// TIA Portal V17 export
// export: Created 2023-12-22T15:28:33.5067968Z, ExportSetting WithDefaults, DisplayName Totally Integrated Automation Portal, DisplayVersion V17, DisplayName TIA Portal Openness, DisplayVersion V17, DisplayName TIA Portal Version Control Interface, DisplayVersion V17, DisplayName STEP 7 Professional, DisplayVersion V17, DisplayName STEP 7 Safety, DisplayVersion V17, DisplayName WinCC Advanced, DisplayVersion V17
DATA_BLOCK "Support_DB"   // DB1000
{ S7_Optimized_Access := 'TRUE' }
VERSION : 0.1
// stored: AutoNumber false, DBAccessibleFromOPCUA true, IsOnlyStoredInLoadMemory false, IsRetainMemResEnabled false, IsWriteProtectedInAS false, MemoryReserve 100
   VAR
      DTR_Clean : Bool;   // Очистка DTR
      DTR_1 : Int;   // Data Transfer 1
      DTR_2 : Int;   // Data Transfer 2
      DTR_3 : Int;   // Data Transfer 3
   END_VAR
   VAR RETAIN
      All_AIs { S7_SetPoint := 'True'} : Int := 399;   // Номер последнего DB аналоговых входов
      All_AOs { S7_SetPoint := 'True'} : Int := 499;   // Номер последнего DB аналоговых выходов
      All_DIs { S7_SetPoint := 'True'} : Int := 209;   // Номер последнего DB дискретных входов
      All_DOs { S7_SetPoint := 'True'} : Int := 219;   // Номер последнего DB дискретных выходов
      All_MDs { S7_SetPoint := 'True'} : Int := 599;   // Номер последнего DB двигателей без ЧП
      All_MDAs { S7_SetPoint := 'True'} : Int := 699;   // Номер последнего DB двигателей с ЧП
      All_VD2s { S7_SetPoint := 'True'} : Int := 799;   // Номер последнего DB заслонки
      All_VD2As { S7_SetPoint := 'True'} : Int := 899;   // Номер последнего DB заслонки с позиционированием
      All_PIDs { S7_SetPoint := 'True'} : Int := 999;   // Номер последнего DB для PID-регулятора
   END_VAR
BEGIN
END_DATA_BLOCK
